{attribute addProperty BoxType "CX5010 EtherCAT slave-1b82-0016"}
{attribute addProperty Id "EMPTY_STRUCTURE"}
{attribute addProperty CRC "0"}
{attribute addProperty SizeInBites "0"}
{attribute addProperty SizeInBytes "0"}
TYPE EMPTY_STRUCTURE :
STRUCT
END_STRUCT
END_TYPE

(* stored: Version 1.2.0.0, ProductVersion 3.1.4024.9
   DUT EMPTY_STRUCTURE: Id {80db4428-d2fc-44e5-a690-d9ddfafa2505} *)
